// TIA Portal V16 export
// export: Created 2022-09-01T14:29:23.5652597Z, ExportSetting WithDefaults, DisplayName Totally Integrated Automation Portal, DisplayVersion V16, DisplayName TIA Portal Version Control Interface, DisplayVersion V16, DisplayName TIA Portal Openness, DisplayVersion V16, DisplayName STEP 7 Professional, DisplayVersion V16, DisplayName STEP 7 Safety, DisplayVersion V16, DisplayName WinCC Advanced, DisplayVersion V16
FUNCTION "Contador_de_Ciclos" : Void   // FC21, LAD
{ S7_Optimized_Access := 'TRUE' }
VERSION : 0.1
// stored: AutoNumber true, IsIECCheckEnabled false, SetENOAutomatically false, UDAEnableTagReadback false
BEGIN

REGION Network 1: Conta o número de ciclos de tratamento
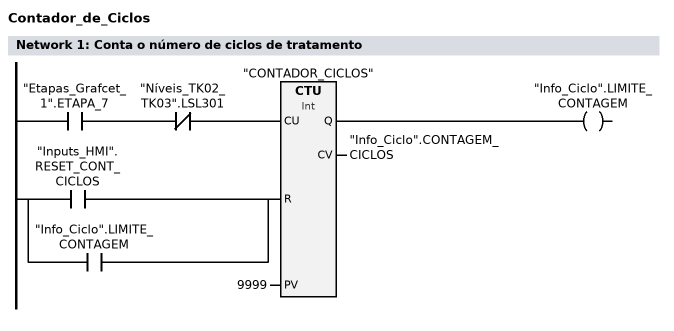
   RUNG wire#powerrail
      Contact( "Etapas_Grafcet_1".ETAPA_7 )
      I_Contact( "Níveis_TK02_TK03".LSL301 )
      { S7_Templates := "value_type := Int" } "CONTADOR_CICLOS".CTU(r := wire#w1, pv := 9999, cv => "Info_Ciclo".CONTAGEM_CICLOS)
      Coil( "Info_Ciclo".LIMITE_CONTAGEM )
   END_RUNG
   RUNG wire#powerrail
      Contact( "Inputs_HMI".RESET_CONT_CICLOS )
   END_RUNG wire#w1
   RUNG wire#powerrail
      Contact( "Info_Ciclo".LIMITE_CONTAGEM )
   END_RUNG wire#w1
   // the same network as SCL:
   "CONTADOR_CICLOS".CTU(CU := "Etapas_Grafcet_1".ETAPA_7 AND NOT "Níveis_TK02_TK03".LSL301,
                         R := "Inputs_HMI".RESET_CONT_CICLOS OR "Info_Ciclo".LIMITE_CONTAGEM,
                         PV := 9999,
                         CV => "Info_Ciclo".CONTAGEM_CICLOS);
   "Info_Ciclo".LIMITE_CONTAGEM := "CONTADOR_CICLOS".Q;
END_REGION
END_FUNCTION
